{attribute 'GeneratedUsingTerminal: EPP5101-0011-0016'}
{attribute addProperty BoxType "EPP5101-0011-0016"}
{attribute addProperty Id "StatusAT %I*Status_D8D782C316Counter_valueAT %I*UINT2Latch_valueAT %I*UINT2"}
{attribute addProperty CRC "2100585715"}
{attribute addProperty Size "20"}
TYPE ENC_Status_compact_7D3464F3 :
STRUCT
	{attribute addProperty Name "Status"}
	Status AT %I* : Status_D8D782C3;
	{attribute addProperty Name "Counter_value"}
	Counter_value AT %I* : UINT;
	{attribute addProperty Name "Latch_value"}
	Latch_value AT %I* : UINT;
END_STRUCT
END_TYPE

(* stored: Version 1.2.0.0, ProductVersion 3.1.4024.9
   DUT ENC_Status_compact_7D3464F3: Id {0b7331e9-d4a5-4ba8-bb9b-a2d47f42a24c} *)
